PROGRAM PRG_Environment
VAR
    {attribute 'TcLinkTo' := 'TIIB[EP2008-0001_M1M2_VCV]^Channel 1^Output'}
    {attribute 'pytmc' := '
        pv: MR1L0:HOMS:VCV
        io: io
        field: ZNAM OFF
        field: ONAM ON
    '}
    bActivateVarCoolMR1L0 AT %Q* : BOOL;
    {attribute 'TcLinkTo' := 'TIIB[EP2008-0001_M1M2_VCV]^Channel 2^Output'}
    {attribute 'pytmc' := '
        pv: MR2L0:HOMS:VCV
        io: io
        field: ZNAM OFF
        field: ONAM ON
    '}
    bActivateVarCoolMR2L0 AT %Q* : BOOL;
END_VAR

    // MR1L0 Flow Pressure Sensors
    GVL_M1L0.fM1L0_Flow_1(iTermBits:=12, fTermMax:=5.0427, fTermMin:=0.050472);
    GVL_M1L0.fM1L0_Flow_1_val := GVL_M1L0.fM1L0_Flow_1.fReal;

    GVL_M1L0.fM1L0_Flow_2(iTermBits:=12, fTermMax:=5.0427, fTermMin:=0.050472);
    GVL_M1L0.fM1L0_Flow_2_val := GVL_M1L0.fM1L0_Flow_2.fReal;

    GVL_M1L0.fM1L0_Press_1(iTermBits:=12, fTermMax:=4.0, fTermMin:=0);
    GVL_M1L0.fM1L0_Press_1_val := GVL_M1L0.fM1L0_Press_1.fReal;

    // MR2L0 Flow Pressure Sensors
    GVL_M2L0.fM2L0_Flow_1(iTermBits:=12, fTermMax:=5.0427, fTermMin:=0.050472);
    GVL_M2L0.fM2L0_Flow_1_val := GVL_M2L0.fM2L0_Flow_1.fReal;

    GVL_M2L0.fM2L0_Flow_2(iTermBits:=12, fTermMax:=5.0427, fTermMin:=0.050472);
    GVL_M2L0.fM2L0_Flow_2_val := GVL_M2L0.fM2L0_Flow_2.fReal;

    GVL_M2L0.fM2L0_Press_1(iTermBits:=12, fTermMax:=4.0, fTermMin:=0);
    GVL_M2L0.fM2L0_Press_1_val := GVL_M2L0.fM2L0_Press_1.fReal;

END_PROGRAM

(* stored: Version 1.1.0.1, ProductVersion 3.1.4022.18
   POU PRG_Environment: Id {ba0070ff-b060-40ec-9097-5e8efb1576b9}, SpecialFunc None *)
